// Chainable 255-character string builder.
FUNCTION_BLOCK FINAL Strb IMPLEMENTS I_Strb
VAR
	_sString	: Str;
	_nLength	: INT;
END_VAR

PROPERTY PRIVATE _this : I_Strb
GET
VAR
	_iThis : I_Strb := THIS^;
END_VAR
_this := _iThis;
END_GET
END_PROPERTY

// Appends text; truncates at 255 chars.
METHOD Append : I_Strb
VAR_INPUT
    sToAdd : Str; // Text to append.
END_VAR

VAR
	_nNewLength	: INT;
END_VAR
Append := _this;

IF sToAdd = '' THEN
	RETURN;
END_IF

_nNewLength := Tc2_Standard.LEN(sToAdd) + _nLength;
IF _nNewLength > 255 THEN
	_nNewLength := 255;
END_IF

_sString := Tc2_Standard.CONCAT(_sString, sToAdd);
_nLength := _nNewLength;
END_METHOD

// Finds first match after position; outputs zero positions when not found.
METHOD FindFirstAfter : I_Strb
VAR_INPUT
    sToFind : Str;      // Text to find.
    nPosition : INT := 1; // One-based start position.
END_VAR
VAR_OUTPUT
    nStart : INT;       // Match start, or 0.
    nEnd : INT;         // Match end, or 0.
END_VAR

VAR
	_sTemp			: Str;
	_nOffset		: INT;
END_VAR
FindFirstAfter := _this;

IF sToFind = '' THEN
	RETURN;
END_IF

IF nPosition = 0 THEN
	RETURN;
END_IF

_sTemp := Tc2_Standard.MID(_sString, _nLength, nPosition);
IF (_nOffset := Tc2_Standard.FIND(_sTemp, sToFind)) <> 0 THEN
	nStart := nPosition + _nOffset - 1;
	nEnd := nPosition + _nOffset - 2 + Tc2_Standard.LEN(sToFind);
END_IF
END_METHOD

// Finds last match before position; outputs zero positions when not found.
METHOD FindLastBefore : I_Strb
VAR_INPUT
    sToFind : Str;        // Text to find.
    nPosition : INT := 256; // One-based end position; 256 means current length.
END_VAR
VAR_OUTPUT
    nStart : INT;         // Match start, or 0.
    nEnd : INT;           // Match end, or 0.
END_VAR
VAR
	_sTemp			: Str;
	_nFindLength	: INT := Tc2_Standard.LEN(sToFind);
	_nOffset		: INT;
END_VAR
FindLastBefore := _this;

IF sToFind = '' THEN
	RETURN;
END_IF

IF nPosition = 0 THEN
	RETURN;
END_IF

IF nPosition = 256 THEN
	nPosition := _nLength;
END_IF

REPEAT
	_sTemp := Tc2_Standard.MID(_sString, _nFindLength, nPosition);
	IF _sTemp = sToFind THEN
		nStart 	:= nPosition;
		nEnd	:= nPosition + _nFindLength - 1;
		RETURN;
	END_IF
UNTIL
	(nPosition := nPosition - 1) <= 0
END_REPEAT
END_METHOD

// Returns current text.
METHOD Get : Str
VAR_INPUT
END_VAR
Get := _sString;
END_METHOD

// Returns current length.
METHOD GetLength : INT
VAR_INPUT
END_VAR
GetLength := _nLength;
END_METHOD

// TRUE when text is found after position.
METHOD HasAfter : BOOL
VAR_INPUT
    sToFind : Str;      // Text to find.
    nPosition : INT := 0; // One-based start position.
END_VAR
VAR_OUTPUT
    nStart : INT;       // Match start, or 0.
    nEnd : INT;         // Match end, or 0.
END_VAR
FindFirstAfter(sToFind, nPosition, nStart => nStart, nEnd => nEnd);
HasAfter := nStart > 0;
END_METHOD

// TRUE when text is found before position.
METHOD HasBefore : BOOL
VAR_INPUT
    sToFind : Str;        // Text to find.
    nPosition : INT := 256; // One-based end position; 256 means current length.
END_VAR
VAR_OUTPUT
    nStart : INT;         // Match start, or 0.
    nEnd : INT;           // Match end, or 0.
END_VAR
IF nPosition = 256 THEN
	nPosition := Tc2_Standard.LEN(_sString);
END_IF

FindLastBefore(sToFind, nPosition, nStart => nStart, nEnd => nEnd);
HasBefore := nStart > 0;
END_METHOD

// Inserts text; no change when position is invalid.
METHOD Inject : I_Strb
VAR_INPUT
    nPosition : INT;    // One-based insert position.
    sToInject : Str;    // Text to insert.
END_VAR
VAR
	_nNewLength	: INT;
END_VAR
Inject := _this;

IF sToInject = '' THEN
	RETURN;
END_IF

IF nPosition = 0 THEN
	RETURN;
END_IF

IF nPosition > _nLength THEN
	RETURN;
END_IF

_nNewLength := Tc2_Standard.LEN(sToInject) + _nLength;
IF _nNewLength > 255 THEN
	_nNewLength := 255;
END_IF

_sString := Tc2_Standard.INSERT(_sString, sToInject, nPosition);
_nLength := _nNewLength;
END_METHOD

// TRUE when current length is 0.
METHOD IsEmpty : BOOL
VAR_INPUT
END_VAR
IsEmpty := _nLength = 0;
END_METHOD

// Outputs current length and returns this builder.
METHOD Length : I_Strb
VAR_OUTPUT
	nLen: INT; // Current length.
END_VAR
Length := _this;
nLen := _nLength;
END_METHOD

// Prepends text; truncates at 255 chars.
METHOD Prepend : I_Strb
VAR_INPUT
    sToAdd : Str; // Text to prepend.
END_VAR
VAR
	_nNewLength	: INT;
END_VAR
Prepend := _this;

IF sToAdd = '' THEN
	RETURN;
END_IF

_nNewLength := Tc2_Standard.LEN(sToAdd) + _nLength;
IF _nNewLength > 255 THEN
	_nNewLength := 255;
END_IF

_sString := Tc2_Standard.CONCAT(sToAdd, _sString);
_nLength := _nNewLength;
END_METHOD

// Removes text; no change when position or length is invalid.
METHOD Remove : I_Strb
VAR_INPUT
    nLength : INT;    // Characters to remove.
    nPosition : INT;  // One-based start position.
END_VAR

VAR
	_nPosition	: INT;
END_VAR
Remove := _this;

IF nPosition = 0 THEN
	RETURN;
END_IF

IF nPosition > _nLength THEN
	RETURN;
END_IF

IF nLength = 0 THEN
	RETURN;
END_IF

IF nLength + nPosition > _nLength THEN
	nLength := _nLength - nPosition + 1;
END_IF

_sString := Tc2_Standard.DELETE(_sString, nLength, nPosition);
_nLength := _nLength - nLength;
END_METHOD

// Sets current text.
METHOD Set : I_Strb
VAR_INPUT
    sValue : Str; // New text.
END_VAR
Set 		:= _this;

_sString 	:= sValue;
_nLength	:= Tc2_Standard.LEN(sValue);
END_METHOD

// Copies substring into sSlice; no change when position or length is invalid.
METHOD Slice : I_Strb
VAR_INPUT
    nLength : INT;   // Characters to copy.
    nPosition : INT; // One-based start position.
END_VAR
VAR_OUTPUT
    sSlice : Strb;   // Output slice builder.
END_VAR
Slice := _this;

IF nPosition = 0 THEN
	RETURN;
END_IF

IF nLength = 0 THEN
	RETURN;
END_IF

sSlice.Set(Tc2_Standard.MID(_sString, nLength, nPosition));
END_METHOD

// Splits text into left and right builders.
METHOD Split : I_Strb
VAR_INPUT
    nPosition : INT; // One-based split position.
END_VAR
VAR_OUTPUT
    sLeft : Strb;    // Left side.
    sRight : Strb;   // Right side.
END_VAR
Split := _this;

IF nPosition = 0 THEN
	RETURN;
END_IF

sLeft.Set(Tc2_Standard.LEFT(_sString, nPosition));
sRight.Set(Tc2_Standard.RIGHT(_sString, _nLength - nPosition));
END_METHOD

// Outputs current text and returns this builder.
METHOD Write : I_Strb;
VAR_OUTPUT
	sOut: Str; // Current text.
END_VAR
Write := _this;
sOut := _sString;
END_METHOD

END_FUNCTION_BLOCK

(* stored: Version 1.1.0.1
   POU Strb: Id {097a9ce5-fff4-459c-bf61-90e104e444f4}, SpecialFunc None
   Folder _: Id {ee5226c4-1bfb-4c78-b582-ae1ec7e3d151}
   Folder I_Build: Id {ac6c8744-50a3-4f05-8763-d0edced1682d}
   Property _this: Id {9f5d4af9-6657-4b84-b94c-f143552d6daa}
   Get Get: Id {57c7bcd7-c66a-4ed8-9ead-784876349f3a}
   Method Append: Id {7f7905f2-7818-4e4d-8188-6df497128569}
   Method FindFirstAfter: Id {8f9e101f-7a2f-44e6-8d32-11ba6ad80cd3}
   Method FindLastBefore: Id {71bc0f49-5ad9-4169-b5ad-3a872c3c466c}
   Method Get: Id {00a5e226-6cad-4cfd-9ed8-2d2605b9d6e6}
   Method GetLength: Id {2dfd9775-4443-406b-99ee-6727c1dce1b5}
   Method HasAfter: Id {f544f3ca-8838-4319-9707-f592713024e1}
   Method HasBefore: Id {62915ef4-82cd-46dc-8a4f-63e40918902b}
   Method Inject: Id {2e9ce33a-9a18-4428-92c8-44eae0f3e5ac}
   Method IsEmpty: Id {9e32988d-1dba-4b45-9469-6ad534af70d9}
   Method Length: Id {43da97c2-f83a-4e05-81ed-ec147eada31a}
   Method Prepend: Id {90cd07b0-8292-43be-8f7c-ccc1f2a79b9d}
   Method Remove: Id {87c2b449-3936-4b9e-bf9e-9a7e13244b52}
   Method Set: Id {4e083d1b-9de2-4451-b0f9-5b881e2173d3}
   Method Slice: Id {41b26e98-f082-480a-832d-cfbb05d20b83}
   Method Split: Id {8062e340-a176-420f-bbf7-07ca296bea0b}
   Method Write: Id {eb0a04ea-d10d-479c-80cd-3778447f4291} *)
